RoboDK station: Visualisering i RoboDK.rdk

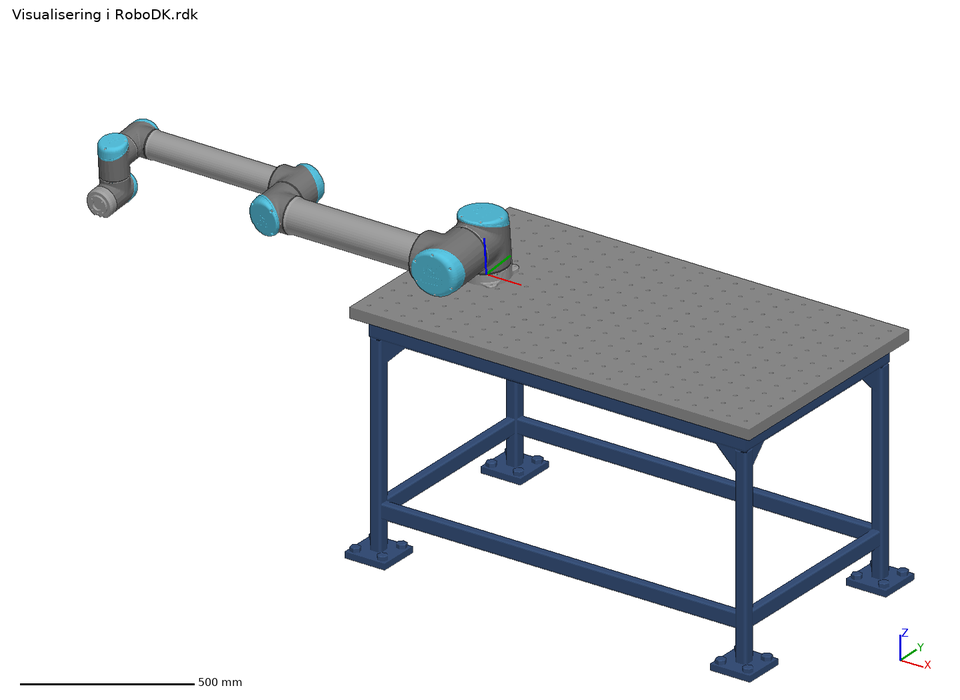
[picture v0: the station drawn from its stored meshes, robots at their saved joint values, targets as dots, program paths as lines]
Station Visualisering i RoboDK (saved by RoboDK 5.5.3). Poses are relative to the parent item; angles as X-Y-Z fixed-axis rotations.
  - frame UR10 Base at (0, 0, 0) mm, rotated rx 5.33 ry 0 rz 0 deg
    - robot UR10: 6 axes, payload 10 kg, reach 1300 mm, repeatability 0.1 mm, weight 28.9 kg
        modified DH rows (alpha deg, a mm, theta deg, d mm): 0, 0, 0, 128; 90, 0, 180, 0; 0, 612.7, 0, 0; 0, 571.6, 0, 163.9; -90, 0, 0, 115.7; 90, 0, 180, 92.2
        joint limits [-360, -360, -360, -360, -360, -360] to [360, 360, 360, 360, 360, 360]; home [0, -90, -90, 0, 90, 0]; saved at [0, 0, -0.171, -0.171, -0.171, -0.171]
  - Python program Wago (listed below)
  - object Table 1400x800x800mm at (140, 0, 0) mm, size 1420 x 820 x 800 mm, geometry from Table-1400x800x800mm.sld

--- Python program Wago ---
import os
import requests
from flask import Flask, jsonify
from flask_mqtt import Mqtt
from robodk.robolink import *  # API to communicate with RoboDK
from robodk.robomath import *  # basic matrix operations

RDK = Robolink()

app = Flask(__name__)

app.config['MQTT_BROKER_URL'] = 'broker.hivemq.com'
app.config['MQTT_BROKER_PORT'] = 1883
app.config['MQTT_USERNAME'] = ''  # Set if necessary
app.config['MQTT_PASSWORD'] = ''  # Set if necessary
app.config['MQTT_KEEPALIVE'] = 5
app.config['MQTT_TLS_ENABLED'] = False

mqtt = Mqtt(app)

robot = RDK.ItemUserPick('Select a robot', ITEM_TYPE_ROBOT)
if not robot.Valid():
    raise Exception('No robot selected or available')

# 1x6 matrix to store the last value for each topic
topic_values = [0, 0, 0, 0, 0, 0]
topic_indices = {
    "triplet/simulator/base": 0,
    "triplet/simulator/shoulder": 1,
    "triplet/simulator/elbow": 2,
    "triplet/simulator/wrist1": 3,
    "triplet/simulator/wrist2": 4,
    "triplet/simulator/wrist3": 5
}

def get_topic_values_request():
    response = requests.get('http://localhost:5000/topic_values')
    if response.status_code == 200:
        return response.json()
    else:
        print(f"Error fetching topic values: {response.status_code}")
        return None

@mqtt.on_connect()
def handle_connect(client, userdata, flags, rc):
    print("Connected with result code " + str(rc))
    for topic in topic_indices.keys():
        mqtt.subscribe(topic)

@mqtt.on_message()
def handle_message(client, userdata, msg):
    topic = msg.topic
    value = msg.payload.decode()
    print(f"Received message '{value}' on topic '{topic}'")

    # Update the value in the topic_values matrix
    index = topic_indices.get(topic)
    if index is not None and topic_values[index] != value:
        topic_values[index] = float(value)
        robot.MoveJ(topic_values)

        # Get the updated topic values
        #updated_values = get_topic_values_request()
        #if updated_values is not None:
            #print(f"Updated topic values: {updated_values}")
            #robot.MoveJ(topic_values)


#@app.route('/topic_values', methods=['GET'])
#def get_topic_values():
    #return (topic_values)

if __name__ == '__main__':
    app.run(debug=False, host="0.0.0.0", port=int(os.environ.get("PORT", 5000)))
